{attribute addProperty BoxType "EK1122-0000-0018"}
{attribute addProperty Id "Beckhoff_EJ5xxxsub_EK1100EK1100_179A0949162"}
{attribute addProperty CRC "121957500"}
{attribute addProperty SizeInBites "16"}
{attribute addProperty SizeInBytes "2"}
TYPE Beckhoff_EJ5xxxEK1122_0744EC7C EXTENDS EK1122_179A0949 :
STRUCT
	{attribute addProperty Name "Beckhoff_EJ5xxxsub_EK1100"}
	Beckhoff_EJ5xxxsub_EK1100 : EK1100_179A0949;
END_STRUCT
END_TYPE

(* stored: Version 1.2.0.0, ProductVersion 3.1.4024.9
   DUT Beckhoff_EJ5xxxEK1122_0744EC7C: Id {12f693ff-6b3b-4f45-bccf-abd98160115f} *)
